FUNCTION_BLOCK PUBLIC ManualControl
VAR_INPUT
	Switch: BOOL;
END_VAR
VAR
	ManualControl: BOOL;
	TimeForInterlockDelay: TIME := T#0.05S;
	ManualMode: BOOL;
	MotorSelection_1: MotorSelection;
	SelectedMotor: INT;
	temp: TIME;
	LowerLeftInterlock: TOF;
	LowerLeft: BOOL;
	LowerRightInterlock: TOF;
	LowerRight: BOOL;
END_VAR
VAR_OUTPUT
	Output: BOOL;
END_VAR
VAR // added by the converter: edge detectors and wires of the graphical bodies
    _w1, _w2, _w3, _w4, _w5 : BOOL;
END_VAR

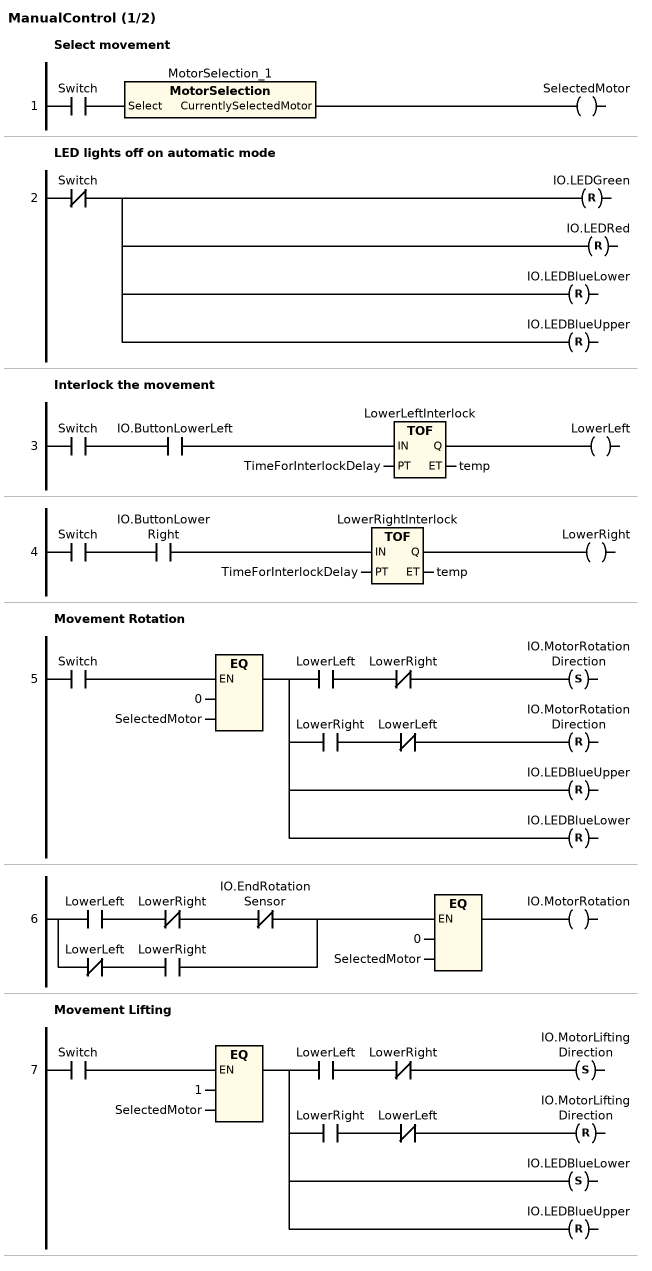
// NETWORK 1: Select movement
MotorSelection_1(Select := Switch); // MotorSelection
SelectedMotor := MotorSelection_1.CurrentlySelectedMotor;

// NETWORK 2: LED lights off on automatic mode
_w1 := NOT Switch;
IO.LEDGreen R= _w1;
IO.LEDRed R= _w1;
IO.LEDBlueLower R= _w1;
IO.LEDBlueUpper R= _w1;

// NETWORK 3: Interlock the movement
LowerLeftInterlock(IN := Switch AND IO.ButtonLowerLeft, PT := TimeForInterlockDelay, ET => temp); // TOF
LowerLeft := LowerLeftInterlock.Q;

// NETWORK 4
LowerRightInterlock(IN := Switch AND IO.ButtonLowerRight, PT := TimeForInterlockDelay, ET => temp); // TOF
LowerRight := LowerRightInterlock.Q;

// NETWORK 5: Movement Rotation
_w2 := Switch AND 0 = SelectedMotor;
IO.MotorRotationDirection S= _w2 AND LowerLeft AND NOT LowerRight;
IO.MotorRotationDirection R= _w2 AND LowerRight AND NOT LowerLeft;
IO.LEDBlueUpper R= _w2;
IO.LEDBlueLower R= _w2;

// NETWORK 6
IO.MotorRotation := (LowerLeft AND NOT LowerRight AND NOT IO.EndRotationSensor OR NOT LowerLeft AND LowerRight) AND 0 = SelectedMotor;

// NETWORK 7: Movement Lifting
_w3 := Switch AND 1 = SelectedMotor;
IO.MotorLiftingDirection S= _w3 AND LowerLeft AND NOT LowerRight;
IO.MotorLiftingDirection R= _w3 AND LowerRight AND NOT LowerLeft;
IO.LEDBlueLower S= _w3;
IO.LEDBlueUpper R= _w3;

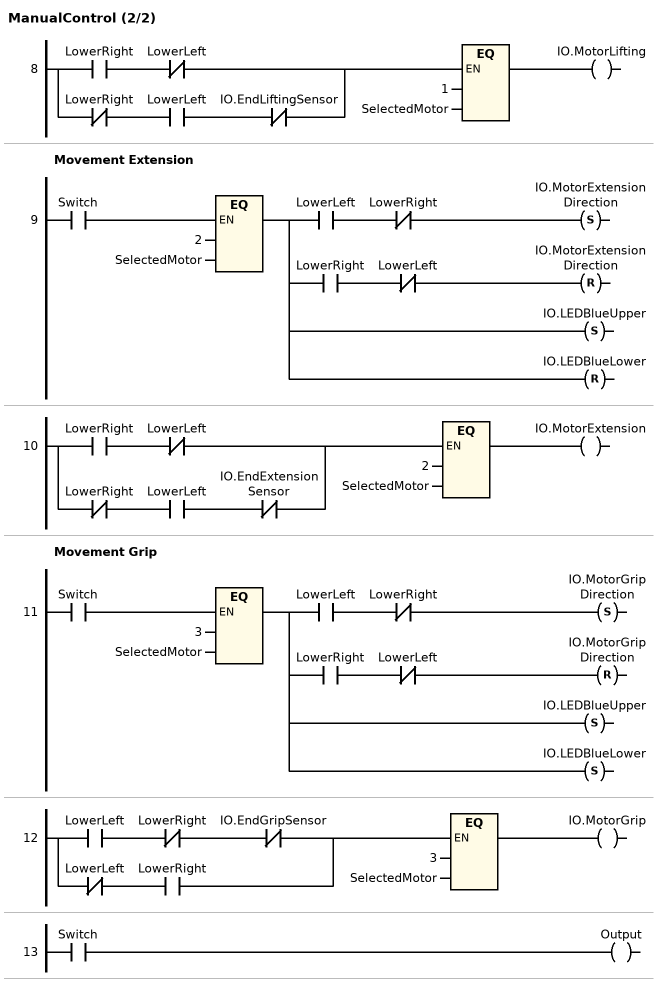
// NETWORK 8
IO.MotorLifting := (LowerRight AND NOT LowerLeft OR NOT LowerRight AND LowerLeft AND NOT IO.EndLiftingSensor) AND 1 = SelectedMotor;

// NETWORK 9: Movement Extension
_w4 := Switch AND 2 = SelectedMotor;
IO.MotorExtensionDirection S= _w4 AND LowerLeft AND NOT LowerRight;
IO.MotorExtensionDirection R= _w4 AND LowerRight AND NOT LowerLeft;
IO.LEDBlueUpper S= _w4;
IO.LEDBlueLower R= _w4;

// NETWORK 10
IO.MotorExtension := (LowerRight AND NOT LowerLeft OR NOT LowerRight AND LowerLeft AND NOT IO.EndExtensionSensor) AND 2 = SelectedMotor;

// NETWORK 11: Movement Grip
_w5 := Switch AND 3 = SelectedMotor;
IO.MotorGripDirection S= _w5 AND LowerLeft AND NOT LowerRight;
IO.MotorGripDirection R= _w5 AND LowerRight AND NOT LowerLeft;
IO.LEDBlueUpper S= _w5;
IO.LEDBlueLower S= _w5;

// NETWORK 12
IO.MotorGrip := (LowerLeft AND NOT LowerRight AND NOT IO.EndGripSensor OR NOT LowerLeft AND LowerRight) AND 3 = SelectedMotor;

// NETWORK 13
Output := Switch;

END_FUNCTION_BLOCK

(* stored: Version 1.1.0.1, ProductVersion 3.1.4024.13
   POU ManualControl: Id {0dc011e3-56d5-4b91-a8d5-8c19aa1fc8c8}, SpecialFunc None *)
